PROGRAM RunGrindingWheel
VAR
END_VAR

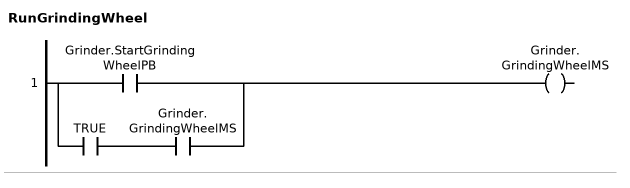
// NETWORK 1
Grinder.GrindingWheelMS := Grinder.StartGrindingWheelPB OR TRUE AND Grinder.GrindingWheelMS;

END_PROGRAM

(* stored: Version 1.1.0.1, ProductVersion 3.1.4024.4
   POU RunGrindingWheel: Id {24c04dbf-19e4-48d1-af90-54bf065a9120}, SpecialFunc None *)
